// TIA Portal project "Loop_Traffic_Light_V1.1" (V18)

(* hardware
DEVICE "S7-1500/ET200MP station_1"  S7-1500 station
   slot 0: "导轨_0"  Rack  6ES7 590-1***0-0AA0
   slot 1: "PLC_1"  CPU 1516-3 PN/DP  6ES7 516-3AN01-0AB0  V2.6
      slot 3: "CPU 显示_1"  6ES7591-1BA00-0AA0
      slot 32768: "PROFINET 接口_1"  X1
      slot 33024: "PROFINET 接口_2"  X2
      slot 33280: "DP 接口_1"  X3
   slot 2: "DI 32x24VDC HF_1"  DI 32x24VDC HF  6ES7 521-1BL00-0AB0  V2.1
   slot 3: "DQ 32x24VDC/0.5A HF_1"  DQ 32x24VDC/0.5A HF  6ES7 522-1BL01-0AB0  V1.1
   slot 4: "AI 8xU/I/RTD/TC ST_1"  AI 8xU/I/RTD/TC ST  6ES7 531-7KF00-0AB0  V2.2
   slot 5: "AQ 4xU/I ST_1"  AQ 4xU/I ST  6ES7 532-5HD00-0AB0  V2.2
DEVICE "HMI_1"  TP700 Comfort
   slot 0: "HMI_1"  TP700 Comfort  6AV2 124-0GC01-0AX0  15.1.0.0
   slot 1: "HMI_RT_1"  TP700 Comfort  6AV2 124-0GC01-0AX0  15.1.0.0
   slot 5: "HMI_1.IE_CP_1"  PROFINET Interface  15.0.1.0
      slot 1: "PROFINET Interface_1"  PROFINET Interface
         slot 1: "Port_1"  Port
         slot 2: "Port_2"  Port
   slot 7: "HMI_1.MPI/DP_CP_1"  MPI/DP Interface  15.0.1.0
*)

// ===== PLC "PLC_1"  CPU 1516-3 PN/DP =====

VAR_GLOBAL   // PLC tag table "默认变量表"
   "System_Byte" AT %MB1 : Byte;
   "FirstScan" AT %M1.0 : Bool;
   "DiagStatusUpdate" AT %M1.1 : Bool;
   "AlwaysTRUE" AT %M1.2 : Bool;
   "AlwaysFALSE" AT %M1.3 : Bool;
   "Clock_Byte" AT %MB0 : Byte;
   "Clock_10Hz" AT %M0.0 : Bool;
   "Clock_5Hz" AT %M0.1 : Bool;
   "Clock_2.5Hz" AT %M0.2 : Bool;
   "Clock_2Hz" AT %M0.3 : Bool;
   "Clock_1.25Hz" AT %M0.4 : Bool;
   "Clock_1Hz" AT %M0.5 : Bool;
   "Clock_0.625Hz" AT %M0.6 : Bool;
   "Clock_0.5Hz" AT %M0.7 : Bool;
   "红灯亮10s" AT %M2.0 : Bool;
   "黄灯亮3s" AT %M2.1 : Bool;
   "绿灯闪烁4s" AT %M2.2 : Bool;
   "红灯" AT %Q1.3 : Bool;
   "循环次数复位" AT %M20.0 : Bool;
   "按钮A" AT %I1.0 : Bool;
   "黄灯" AT %Q1.2 : Bool;
   "绿灯" AT %Q1.1 : Bool;
   "按钮B" AT %I1.1 : Bool;
   "循环次数" AT %MW100 : Word;
   "Tag_1" AT %M10.0 : Bool;
END_VAR

DATA_BLOCK "红绿灯循环逻辑_DB"   // DB1
{ S7_Optimized_Access := 'TRUE' }
VERSION : 0.1
// stored: InstanceOfName 红绿灯循环逻辑
"红绿灯循环逻辑"
BEGIN
END_DATA_BLOCK

DATA_BLOCK "全局DB"   // DB8
{ S7_Optimized_Access := 'TRUE' }
VERSION : 0.1
   VAR
      循环次数 : DInt;
      启动 : Bool;   // 按钮A
      停止 : Bool;   // 按钮B
      灯状态 : DInt;
   END_VAR
BEGIN
END_DATA_BLOCK

FUNCTION_BLOCK "红绿灯循环逻辑"   // FB1, LAD
{ S7_Optimized_Access := 'TRUE' }
VERSION : 0.1
   VAR
      C1 : IEC_COUNTER;
      红灯 : "红灯逻辑";
      黄灯 : "黄灯逻辑";
      绿灯 : "绿灯逻辑";
      红灯状态 : DInt;
      黄灯状态 : DInt;
      绿灯状态 : DInt;
   END_VAR
BEGIN

REGION Network 1: 按钮A
   // 不自锁发现HMI按钮按了根本没用www
   // 
   // 现在主要是说吧红灯维持在0和1
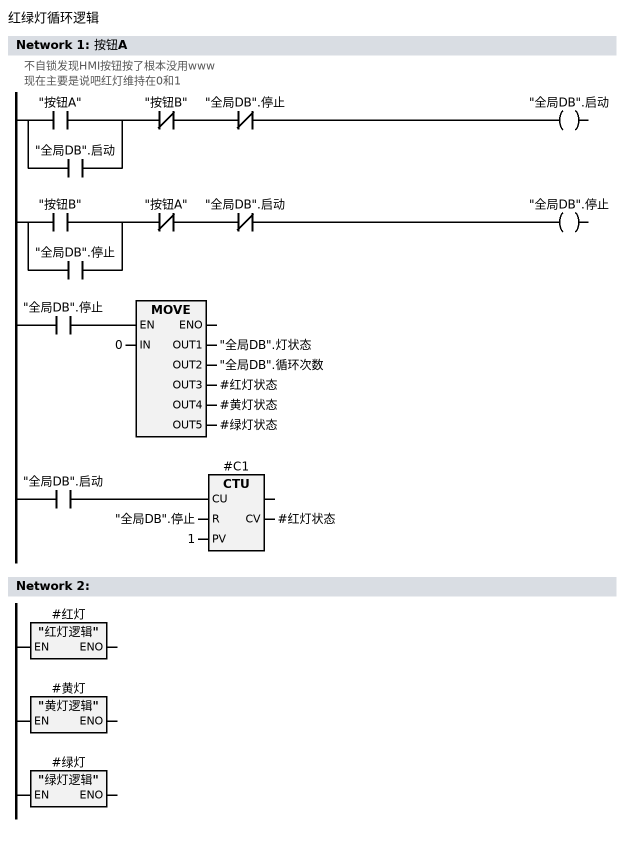
   "全局DB".启动 := ("按钮A" OR "全局DB".启动) AND NOT "按钮B" AND NOT "全局DB".停止;
   "全局DB".停止 := ("按钮B" OR "全局DB".停止) AND NOT "按钮A" AND NOT "全局DB".启动;
   IF "全局DB".停止 THEN
       "全局DB".灯状态 := 0;
       "全局DB".循环次数 := 0;
       #红灯状态 := 0;
       #黄灯状态 := 0;
       #绿灯状态 := 0;
   END_IF;
   #C1.CTU(CU := "全局DB".启动, R := "全局DB".停止, PV := 1, CV => #红灯状态);
END_REGION

REGION Network 2
   RUNG wire#powerrail
      #红灯()
   END_RUNG
   RUNG wire#powerrail
      #黄灯()
   END_RUNG
   RUNG wire#powerrail
      #绿灯()
   END_RUNG
   // the same network as SCL:
   #红灯();   // "红灯逻辑"
   #黄灯();   // "黄灯逻辑"
   #绿灯();   // "绿灯逻辑"
END_REGION
END_FUNCTION_BLOCK

FUNCTION_BLOCK "红灯逻辑"   // FB2, LAD
{ S7_Optimized_Access := 'TRUE' }
VERSION : 0.1
   VAR
      TON_DB : IEC_TIMER;
   END_VAR
   VAR_TEMP   // added for the SCL form of the ladder/FBD networks
      _w1 : Bool;
   END_VAR
BEGIN

REGION Network 1
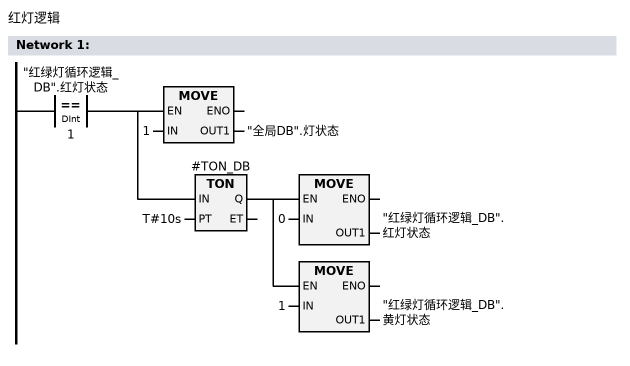
   #_w1 := "红绿灯循环逻辑_DB".红灯状态 = 1;
   IF #_w1 THEN "全局DB".灯状态 := 1; END_IF;
   #TON_DB.TON(IN := #_w1, PT := T#10s);
   IF #TON_DB.Q THEN
       "红绿灯循环逻辑_DB".红灯状态 := 0;
       "红绿灯循环逻辑_DB".黄灯状态 := 1;
   END_IF;
END_REGION
END_FUNCTION_BLOCK

FUNCTION_BLOCK "黄灯逻辑"   // FB3, LAD
{ S7_Optimized_Access := 'TRUE' }
VERSION : 0.1
   VAR
      TON_DB : IEC_TIMER;
   END_VAR
   VAR_TEMP   // added for the SCL form of the ladder/FBD networks
      _w1 : Bool;
   END_VAR
BEGIN

REGION Network 1
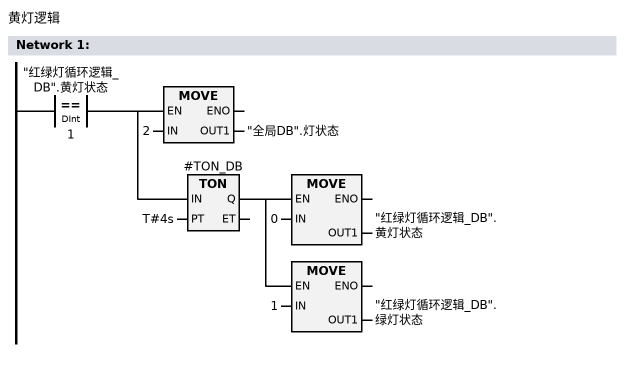
   #_w1 := "红绿灯循环逻辑_DB".黄灯状态 = 1;
   IF #_w1 THEN "全局DB".灯状态 := 2; END_IF;
   #TON_DB.TON(IN := #_w1, PT := T#4s);
   IF #TON_DB.Q THEN
       "红绿灯循环逻辑_DB".黄灯状态 := 0;
       "红绿灯循环逻辑_DB".绿灯状态 := 1;
   END_IF;
END_REGION
END_FUNCTION_BLOCK

FUNCTION_BLOCK "绿灯逻辑"   // FB4, LAD
{ S7_Optimized_Access := 'TRUE' }
VERSION : 0.1
   VAR
      TON_DB : IEC_TIMER;
      CTU_DB : IEC_DCOUNTER;
   END_VAR
   VAR_TEMP   // added for the SCL form of the ladder/FBD networks
      _w1 : Bool;
   END_VAR
BEGIN

REGION Network 1
   // 难道说INC放后面,就不会说因为INC一直执行而MOVE不运行?
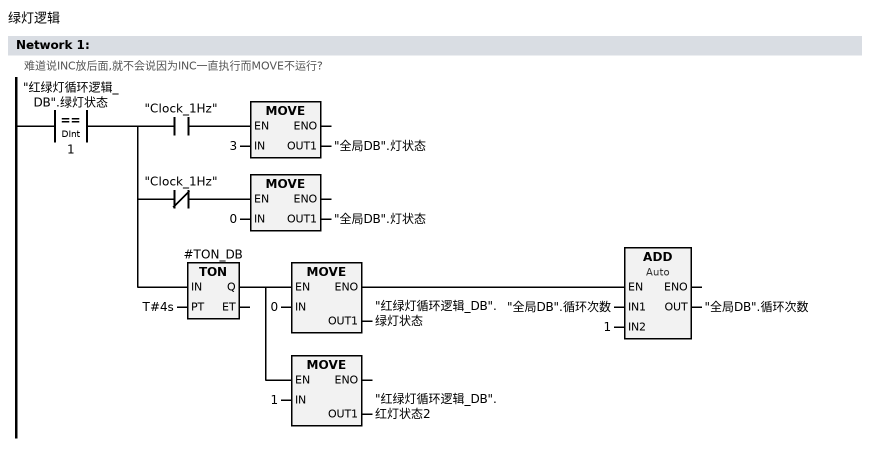
   #_w1 := "红绿灯循环逻辑_DB".绿灯状态 = 1;
   IF #_w1 AND "Clock_1Hz" THEN "全局DB".灯状态 := 3; END_IF;
   IF #_w1 AND NOT "Clock_1Hz" THEN "全局DB".灯状态 := 0; END_IF;
   #TON_DB.TON(IN := #_w1, PT := T#4s);
   IF #TON_DB.Q THEN
       "红绿灯循环逻辑_DB".绿灯状态 := 0;
       "全局DB".循环次数 := "全局DB".循环次数 + 1;
       "红绿灯循环逻辑_DB".红灯状态2 := 1;
   END_IF;
END_REGION
END_FUNCTION_BLOCK

ORGANIZATION_BLOCK "Main"   // OB1, LAD, ProgramCycle
TITLE = "Main Program Sweep (Cycle)"
{ S7_Optimized_Access := 'TRUE' }
VERSION : 0.1
   VAR_INPUT
      Initial_Call : Bool;   // Initial call of this OB
      Remanence : Bool;   // =True, if remanent data are available
   END_VAR
BEGIN

REGION Network 1
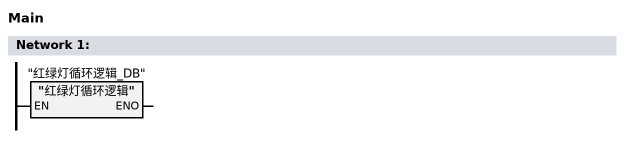
   RUNG wire#powerrail
      "红绿灯循环逻辑_DB"()
   END_RUNG
   // the same network as SCL:
   "红绿灯循环逻辑_DB"();   // "红绿灯循环逻辑"
END_REGION

REGION Network 2
   // 黄灯
END_REGION

REGION Network 3
   // 绿灯
END_REGION
END_ORGANIZATION_BLOCK

(* ===== HMI "HMI_RT_1" =====
system functions are stored by id; their names below are inferred from use
connection "HMI_连接_1": ETHERNET, S7_1500_OMS

HMI tags "默认变量表"
   "Tag_ScreenNumber" : UInt, internal
   "全局DB_循环次数" : DInt = PLC 全局DB.循环次数, 100 ms
   "全局DB_启动" : Bool = PLC 全局DB.启动, 100 ms
   "全局DB_停止" : Bool = PLC 全局DB.停止, 100 ms
   "全局DB_灯状态" : DInt = PLC 全局DB.灯状态, 100 ms

screen "根画面" 800x420, template "模板_1"
   on GenerateScreen: SetTag("Tag_ScreenNumber", 1)
   Button "按钮_1" at 133,71 size 156x67; TextOff '按钮A'
      on Press: SetBit("全局DB_启动")
      on Release: ResetBit("全局DB_启动")
   Button "按钮_2" at 133,143 size 156x75; TextOff '按钮B'
      on Release: ResetBit("全局DB_停止")
      on Press: SetBit("全局DB_停止")
   Circle "圆_1" at 456,73 size 48x48
      Appearance <- "全局DB_灯状态"
   IOField "I/O 域_1" at 418,146 size 115x43; FormatPattern 99999
      ProcessValue <- "全局DB_循环次数"
   TextField "文本域_4" at 553,162 size 73x20; Text '循环次数'

Template "模板_1" 800x420
   Button "退出" at 720,360 size 78x58; TextOff '退出'; PictureOff "ExitRuntime_TP700_Comfort_TR"; PictureOn "ExitRuntime_TP700_Comfort_TR"
      on Release: StopRuntime(0)
   Button "Template_Button" at 640,360 size 78x58; TextOff 'Text'
   Button "Template_Button_1" at 560,360 size 78x58; TextOff 'Text'
   Button "Template_Button_2" at 480,360 size 78x58; TextOff 'Text'
   Button "Template_Button_3" at 400,360 size 78x58; TextOff 'Text'
   Button "Template_Button_4" at 321,360 size 78x58; TextOff 'Text'
   Button "Template_Button_5" at 241,360 size 78x58; TextOff 'Text'
   Button "Template_Button_6" at 161,360 size 78x58; TextOff 'Text'
   Button "报警" at 81,360 size 78x58; TextOff '报警'; PictureOff "AlarmDisplay_TP700_Comfort_TR"; PictureOn "AlarmDisplay_TP700_Comfort_TR"
      on Release: function_ef3f5d25("报警窗口_Unacknowledged", -1)
   Button "起始画面" at 1,360 size 78x58; TextOff '起始画面'; PictureOff "NavigateHome_TP700_Comfort_TR"; PictureOn "NavigateHome_TP700_Comfort_TR"
      on Release: ActivateScreen("根画面", 0)
*)